// TIA Portal project "Soru5" (V15)

(* hardware
DEVICE "S7-1200 station_1"  S7-1200 Station
   slot 0: "Rack_0"  S7-1200 Rack  Rack  V1.0
   slot 1: "PLC_1"  CPU 1214C DC/DC/DC  6ES7 214-1AG40-0XB0  V4.2
*)

// ===== PLC "PLC_1"  CPU 1214C DC/DC/DC =====

VAR_GLOBAL   // PLC tag table "Default tag table"
   "Dudur" AT %I0.0 : Bool;
   "Baslat" AT %I0.1 : Bool;
   "Yıldız" AT %Q0.0 : Bool;
   "Ucgen" AT %Q0.1 : Bool;
   "DCfren" AT %Q0.2 : Bool;
END_VAR

// folder: System blocks/Program resources

DATA_BLOCK "zmn"   // DB1
{ S7_Optimized_Access := 'TRUE' }
AUTHOR : Simatic
FAMILY : IEC
NAME : IEC_TMR
VERSION : 1.0
// stored: InstanceOfName IEC_TIMER
"IEC_TIMER"
BEGIN
END_DATA_BLOCK

// folder: (top level)

ORGANIZATION_BLOCK "Main"   // OB1, LAD, ProgramCycle
TITLE = "Main Program Sweep (Cycle)"
{ S7_Optimized_Access := 'TRUE' }
VERSION : 0.1
   VAR_INPUT
      Initial_Call : Bool;   // Initial call of this OB
      Remanence : Bool;   // =True, if remanent data are available
   END_VAR
BEGIN

REGION Network 1: Yıdızda üçgene geçme için zamanlayıcı rölesi
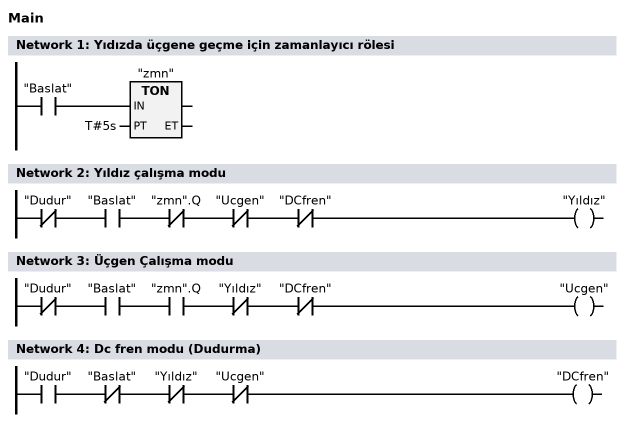
   "zmn".TON(IN := "Baslat", PT := T#5s);
END_REGION

REGION Network 2: Yıldız çalışma modu
   RUNG wire#powerrail
      I_Contact( "Dudur" )
      Contact( "Baslat" )
      I_Contact( "zmn".Q )
      I_Contact( "Ucgen" )
      I_Contact( "DCfren" )
      Coil( "Yıldız" )
   END_RUNG
   // the same network as SCL:
   "Yıldız" := NOT "Dudur" AND "Baslat" AND NOT "zmn".Q AND NOT "Ucgen" AND NOT "DCfren";
END_REGION

REGION Network 3: Üçgen Çalışma modu
   RUNG wire#powerrail
      I_Contact( "Dudur" )
      Contact( "Baslat" )
      Contact( "zmn".Q )
      I_Contact( "Yıldız" )
      I_Contact( "DCfren" )
      Coil( "Ucgen" )
   END_RUNG
   // the same network as SCL:
   "Ucgen" := NOT "Dudur" AND "Baslat" AND "zmn".Q AND NOT "Yıldız" AND NOT "DCfren";
END_REGION

REGION Network 4: Dc fren modu (Dudurma)
   RUNG wire#powerrail
      Contact( "Dudur" )
      I_Contact( "Baslat" )
      I_Contact( "Yıldız" )
      I_Contact( "Ucgen" )
      Coil( "DCfren" )
   END_RUNG
   // the same network as SCL:
   "DCfren" := "Dudur" AND NOT "Baslat" AND NOT "Yıldız" AND NOT "Ucgen";
END_REGION
END_ORGANIZATION_BLOCK